# B&R Automation Studio project TD52 (part 67)

```c
  /* InitializeConditions for Delay: '<S15>/Resettable Delay' */
  Gen2_ref_DWork->icLoad_nl = true;

  /* InitializeConditions for Delay: '<Root>/Delay2' */
  Gen2_ref_DWork->icLoad_e = true;

  /* InitializeConditions for DiscreteIntegrator: '<S760>/Discrete-Time Integrator' */
  Gen2_ref_DWork->DiscreteTimeIntegrator_DSTATE_h = 1.0;

  /* InitializeConditions for Delay: '<S795>/Delay' */
  Gen2_ref_DWork->icLoad_h = true;

  /* InitializeConditions for DiscreteIntegrator: '<S579>/Discrete-Time Integrator' */
  Gen2_ref_DWork->DiscreteTimeIntegrator_DSTATE_m = 1.7;

  /* InitializeConditions for UnitDelay: '<S14>/Unit Delay4' */
  Gen2_ref_DWork->UnitDelay4_DSTATE_d = true;

  /* InitializeConditions for Delay: '<S14>/Resettable Delay2' */
  Gen2_ref_DWork->icLoad_l = true;

  /* InitializeConditions for Delay: '<S14>/Resettable Delay' */
  Gen2_ref_DWork->icLoad_i = true;

  /* InitializeConditions for UnitDelay: '<S14>/Unit Delay' */
  Gen2_ref_DWork->UnitDelay_DSTATE = 1.7;

  /* InitializeConditions for Delay: '<S14>/Resettable Delay3' */
  Gen2_ref_DWork->icLoad_f = true;

  /* InitializeConditions for DiscreteIntegrator: '<S748>/Discrete-Time Integrator' */
  Gen2_ref_DWork->DiscreteTimeIntegrator_IC_LOADI = 1U;

  /* InitializeConditions for DiscreteIntegrator: '<S748>/Discrete-Time Integrator4' */
  Gen2_ref_DWork->DiscreteTimeIntegrator4_DSTATE = 0.0;
  if (Gen2_ref_DWork->DiscreteTimeIntegrator4_DSTATE >= 0.0) {
    Gen2_ref_DWork->DiscreteTimeIntegrator4_DSTATE = 0.0;
  } else if (Gen2_ref_DWork->DiscreteTimeIntegrator4_DSTATE <= -0.3) {
    Gen2_ref_DWork->DiscreteTimeIntegrator4_DSTATE = -0.3;
  }

  /* End of InitializeConditions for DiscreteIntegrator: '<S748>/Discrete-Time Integrator4' */

  /* InitializeConditions for Delay: '<S637>/Resettable Delay' */
  Gen2_ref_DWork->icLoad_ef = true;

  /* InitializeConditions for Delay: '<S637>/Variable Integer Delay' */
  Gen2_ref_DWork->icLoad_b = true;

  /* InitializeConditions for UnitDelay: '<S628>/Unit Delay1' */
  Gen2_ref_DWork->UnitDelay1_DSTATE_a = 1.0;

  /* InitializeConditions for Delay: '<S625>/Delay' */
  Gen2_ref_DWork->Delay_DSTATE_k = 287.0;

  /* InitializeConditions for Delay: '<S666>/Resettable Delay' */
  Gen2_ref_DWork->icLoad_i0 = true;

  /* InitializeConditions for Delay: '<S714>/Resettable Delay1' */
  Gen2_ref_DWork->icLoad_np = true;

  /* InitializeConditions for Delay: '<S714>/Resettable Delay' */
  Gen2_ref_DWork->icLoad_j = true;

  /* InitializeConditions for Delay: '<S715>/Resettable Delay1' */
  Gen2_ref_DWork->icLoad_a = true;

  /* InitializeConditions for Delay: '<S715>/Resettable Delay' */
  Gen2_ref_DWork->icLoad_m3 = true;

  /* InitializeConditions for Delay: '<S431>/Delay' */
  Gen2_ref_DWork->icLoad_b3 = true;

  /* InitializeConditions for Delay: '<S78>/Variable Integer Delay' */
  Gen2_ref_DWork->icLoad_ev = true;

  /* InitializeConditions for Delay: '<S88>/Delay' */
  Gen2_ref_DWork->icLoad_d = true;

  /* InitializeConditions for Delay: '<S90>/Delay' */
  Gen2_ref_DWork->icLoad_es = true;

  /* InitializeConditions for Delay: '<S87>/Delay' */
  Gen2_ref_DWork->icLoad_evr = true;

  /* InitializeConditions for Delay: '<S89>/Delay' */
  Gen2_ref_DWork->icLoad_fg = true;

  /* InitializeConditions for Delay: '<S77>/Variable Integer Delay' */
  Gen2_ref_DWork->icLoad_c = true;

  /* InitializeConditions for Delay: '<S80>/Delay' */
  Gen2_ref_DWork->icLoad_eu = true;

  /* InitializeConditions for Delay: '<S82>/Delay' */
  Gen2_ref_DWork->icLoad_ee = true;

  /* InitializeConditions for Delay: '<S79>/Delay' */
  Gen2_ref_DWork->icLoad_ki = true;

  /* InitializeConditions for Delay: '<S81>/Delay' */
  Gen2_ref_DWork->icLoad_h3 = true;

  /* InitializeConditions for UnitDelay: '<S53>/Unit Delay4' */
  Gen2_ref_DWork->UnitDelay4_DSTATE_o = true;

  /* InitializeConditions for Delay: '<S63>/Delay' */
  Gen2_ref_DWork->icLoad_g = true;

  /* InitializeConditions for Delay: '<S64>/Delay' */
  Gen2_ref_DWork->icLoad_c1 = true;

  /* InitializeConditions for UnitDelay: '<S23>/Unit Delay3' */
  Gen2_ref_DWork->UnitDelay3_DSTATE_gf = true;

  /* InitializeConditions for DiscreteIntegrator: '<S132>/Discrete-Time Integrator' */
  Gen2_ref_DWork->DiscreteTimeIntegrator_DSTATE_g = 100000.0;

  /* InitializeConditions for Delay: '<S45>/Delay' */
  Gen2_ref_DWork->icLoad_eh = true;

  /* InitializeConditions for Delay: '<S161>/Delay2' */
  Gen2_ref_DWork->Delay2_DSTATE_f = true;

  /* InitializeConditions for DiscreteIntegrator: '<S45>/Discrete-Time Integrator1' */
  Gen2_ref_DWork->DiscreteTimeIntegrator1_IC_LOAD = 1U;

  /* InitializeConditions for Delay: '<S26>/Delay' */
  Gen2_ref_DWork->icLoad_kq = true;

  /* InitializeConditions for Delay: '<S111>/Delay2' */
  Gen2_ref_DWork->Delay2_DSTATE_k = true;

  /* InitializeConditions for DiscreteIntegrator: '<S26>/Discrete-Time Integrator' */
  Gen2_ref_DWork->DiscreteTimeIntegrator_IC_LOA_l = 1U;

  /* InitializeConditions for Delay: '<S494>/Delay' */
  Gen2_ref_DWork->icLoad_ir = true;

  /* InitializeConditions for Delay: '<S708>/Delay' */
  Gen2_ref_DWork->icLoad_nv = true;

  /* InitializeConditions for Delay: '<S524>/Delay' */
  Gen2_ref_DWork->icLoad_dk = true;

  /* InitializeConditions for Delay: '<S811>/Delay' */
  Gen2_ref_DWork->icLoad_iv = true;

  /* InitializeConditions for Delay: '<S830>/Resettable Delay' */
  Gen2_ref_DWork->icLoad_ix = true;

  /* InitializeConditions for Delay: '<S830>/Delay' */
  Gen2_ref_DWork->Delay_DSTATE_n2 = true;

  /* InitializeConditions for Delay: '<S666>/Delay' */
  Gen2_ref_DWork->Delay_DSTATE_cnq = true;

  /* InitializeConditions for Delay: '<S714>/Delay' */
  Gen2_ref_DWork->Delay_DSTATE_a = true;

  /* InitializeConditions for Delay: '<S715>/Delay' */
  Gen2_ref_DWork->Delay_DSTATE_ng = true;

  /* SystemInitialize for Atomic SubSystem: '<S418>/2nd Order Filter' */
  Gen2_ref_undOrderFilter3_Init(&Gen2_ref_DWork->undOrderFilter_j, inst);

  /* End of SystemInitialize for SubSystem: '<S418>/2nd Order Filter' */

  /* SystemInitialize for Atomic SubSystem: '<S418>/Filter' */
  /* InitializeConditions for DiscreteIntegrator: '<S439>/Discrete-Time Integrator' */
  Gen2_ref_DWork->DiscreteTimeIntegrator_IC_LOA_f = 1U;

  /* End of SystemInitialize for SubSystem: '<S418>/Filter' */

  /* SystemInitialize for Atomic SubSystem: '<S201>/Volt_filt' */
  Gen2_ref_N_TC_HP_filt_Init(&Gen2_ref_DWork->Volt_filt, inst);

  /* End of SystemInitialize for SubSystem: '<S201>/Volt_filt' */

  /* SystemInitialize for Atomic SubSystem: '<S205>/p2s_filt' */
  Gen2_ref_N_TC_HP_filt_Init(&Gen2_ref_DWork->p2s_filt, inst);

  /* End of SystemInitialize for SubSystem: '<S205>/p2s_filt' */

  /* SystemInitialize for Atomic SubSystem: '<S425>/TOF' */
  Gen2_ref_TOF_Init(&Gen2_ref_DWork->TOF_h, inst);

  /* End of SystemInitialize for SubSystem: '<S425>/TOF' */

  /* SystemInitialize for Atomic SubSystem: '<S425>/Filter' */
  /* InitializeConditions for DiscreteIntegrator: '<S485>/Discrete-Time Integrator' */
  Gen2_ref_DWork->DiscreteTimeIntegrator_IC_LOA_p = 1U;

  /* End of SystemInitialize for SubSystem: '<S425>/Filter' */

  /* SystemInitialize for Atomic SubSystem: '<S427>/TOF1' */
  Gen2_ref_TOF_Init(&Gen2_ref_DWork->TOF1_o, inst);

  /* End of SystemInitialize for SubSystem: '<S427>/TOF1' */

  /* SystemInitialize for Atomic SubSystem: '<S427>/TP' */
  Gen2_ref_TP_Init(&Gen2_ref_DWork->TP_p, inst);

  /* End of SystemInitialize for SubSystem: '<S427>/TP' */

  /* SystemInitialize for Atomic SubSystem: '<S345>/p2sfilt' */
  Gen2_ref_N_TC_HP_filt_Init(&Gen2_ref_DWork->p2sfilt, inst);

  /* End of SystemInitialize for SubSystem: '<S345>/p2sfilt' */

  /* SystemInitialize for Atomic SubSystem: '<S194>/Pel_filt' */
  Gen2_ref_N_TC_HP_filt_Init(&Gen2_ref_DWork->Pel_filt, inst);

  /* End of SystemInitialize for SubSystem: '<S194>/Pel_filt' */

  /* SystemInitialize for Atomic SubSystem: '<S875>/Pd_filt' */
  Gen2_ref_Pd_filt_Init(&Gen2_ref_DWork->Pd_filt_p, inst);

  /* End of SystemInitialize for SubSystem: '<S875>/Pd_filt' */

  /* SystemInitialize for Atomic SubSystem: '<S344>/Pd_filt' */
  Gen2_ref_Pd_filt_Init(&Gen2_ref_DWork->Pd_filt, inst);

  /* End of SystemInitialize for SubSystem: '<S344>/Pd_filt' */

  /* SystemInitialize for Atomic SubSystem: '<S344>/WO1' */
  Gen2_ref_Filter1_Init(&Gen2_ref_DWork->WO1, inst);

  /* End of SystemInitialize for SubSystem: '<S344>/WO1' */

  /* SystemInitialize for Atomic SubSystem: '<S344>/WO2' */
  Gen2_ref_Filter3_Init(Gen2_ref_ConstB.tde1, &Gen2_ref_DWork->WO2, inst);

  /* End of SystemInitialize for SubSystem: '<S344>/WO2' */

  /* SystemInitialize for Atomic SubSystem: '<S190>/N_TC_HP_filt' */
  Gen2_ref_N_TC_HP_filt_Init(&Gen2_ref_DWork->N_TC_HP_filt, inst);

  /* End of SystemInitialize for SubSystem: '<S190>/N_TC_HP_filt' */

  /* SystemInitialize for Atomic SubSystem: '<S197>/T2s_filt' */
  Gen2_ref_N_TC_HP_filt_Init(&Gen2_ref_DWork->T2s_filt, inst);

  /* End of SystemInitialize for SubSystem: '<S197>/T2s_filt' */

  /* SystemInitialize for Atomic SubSystem: '<S193>/N_TC_LP_filt' */
  Gen2_ref_N_TC_HP_filt_Init(&Gen2_ref_DWork->N_TC_LP_filt_f, inst);

  /* End of SystemInitialize for SubSystem: '<S193>/N_TC_LP_filt' */

  /* SystemInitialize for Atomic SubSystem: '<S19>/Filter1' */
  Gen2_ref_Filter3_Init(1.0, &Gen2_ref_DWork->Filter1_l, inst);

  /* End of SystemInitialize for SubSystem: '<S19>/Filter1' */

  /* SystemInitialize for Atomic SubSystem: '<S6>/TOF' */
  Gen2_ref_TOF_Init(&Gen2_ref_DWork->TOF, inst);

  /* End of SystemInitialize for SubSystem: '<S6>/TOF' */

  /* SystemInitialize for Atomic SubSystem: '<S6>/TOF1' */
  Gen2_ref_TOF_Init(&Gen2_ref_DWork->TOF1, inst);

  /* End of SystemInitialize for SubSystem: '<S6>/TOF1' */

  /* SystemInitialize for Atomic SubSystem: '<S6>/TOF2' */
  Gen2_ref_TOF_Init(&Gen2_ref_DWork->TOF2, inst);

  /* End of SystemInitialize for SubSystem: '<S6>/TOF2' */

  /* SystemInitialize for Atomic SubSystem: '<S343>/PID_Power' */
  /* InitializeConditions for DiscreteIntegrator: '<S389>/Discrete-Time Integrator' */
  Gen2_ref_DWork->DiscreteTimeIntegrator_IC_LOA_c = 1U;

  /* InitializeConditions for Delay: '<S394>/Delay' */
  Gen2_ref_DWork->icLoad_ht = true;

  /* End of SystemInitialize for SubSystem: '<S343>/PID_Power' */

  /* SystemInitialize for Atomic SubSystem: '<S760>/p2sfilt' */
  Gen2_ref_N_TC_HP_filt_Init(&Gen2_ref_DWork->p2sfilt_l, inst);

  /* End of SystemInitialize for SubSystem: '<S760>/p2sfilt' */

  /* SystemInitialize for Atomic SubSystem: '<S424>/speed Filter' */
  Gen2_ref_N_TC_HP_filt_Init(&Gen2_ref_DWork->speedFilter, inst);

  /* End of SystemInitialize for SubSystem: '<S424>/speed Filter' */

  /* SystemInitialize for Atomic SubSystem: '<S424>/Filter1' */
  Gen2_ref_Filter1_Init(&Gen2_ref_DWork->Filter1_f, inst);

  /* End of SystemInitialize for SubSystem: '<S424>/Filter1' */

  /* SystemInitialize for Atomic SubSystem: '<S761>/Filter1' */
  Gen2_ref_Filter3_Init(Gen2_ref_ConstB.Constant1_g, &Gen2_ref_DWork->Filter1_p, inst);

  /* End of SystemInitialize for SubSystem: '<S761>/Filter1' */

  /* SystemInitialize for Atomic SubSystem: '<S761>/Filter' */
  Gen2_ref_Pd_filt_Init(&Gen2_ref_DWork->Filter_kj, inst);

  /* End of SystemInitialize for SubSystem: '<S761>/Filter' */

  /* SystemInitialize for Atomic SubSystem: '<S585>/Filter1' */
  Gen2_ref_N_TC_HP_filt_Init(&Gen2_ref_DWork->Filter1_fg, inst);

  /* End of SystemInitialize for SubSystem: '<S585>/Filter1' */

  /* SystemInitialize for Atomic SubSystem: '<S585>/Filter' */
  Gen2_ref_Filter3_Init(1.0, &Gen2_ref_DWork->Filter_n, inst);

  /* End of SystemInitialize for SubSystem: '<S585>/Filter' */

  /* SystemInitialize for Atomic SubSystem: '<S306>/2nd Order Filter' */
  Gen2_ref_undOrderFilter_Init(&Gen2_ref_DWork->undOrderFilter, inst);

  /* End of SystemInitialize for SubSystem: '<S306>/2nd Order Filter' */

  /* SystemInitialize for Atomic SubSystem: '<S306>/2nd Order Filter1' */
  Gen2_ref_undOrderFilter_Init(&Gen2_ref_DWork->undOrderFilter1, inst);

  /* End of SystemInitialize for SubSystem: '<S306>/2nd Order Filter1' */

  /* SystemInitialize for Atomic SubSystem: '<S306>/2nd Order Filter2' */
  Gen2_ref_undOrderFilter_Init(&Gen2_ref_DWork->undOrderFilter2, inst);

  /* End of SystemInitialize for SubSystem: '<S306>/2nd Order Filter2' */

  /* SystemInitialize for Atomic SubSystem: '<S306>/2nd Order Filter3' */
  Gen2_ref_undOrderFilter3_Init(&Gen2_ref_DWork->undOrderFilter3, inst);

  /* End of SystemInitialize for SubSystem: '<S306>/2nd Order Filter3' */

  /* SystemInitialize for Atomic SubSystem: '<S196>/T1LP_filt' */
  Gen2_ref_N_TC_HP_filt_Init(&Gen2_ref_DWork->T1LP_filt, inst);

  /* End of SystemInitialize for SubSystem: '<S196>/T1LP_filt' */

  /* SystemInitialize for Atomic SubSystem: '<S195>/T1HP_filt' */
  Gen2_ref_N_TC_HP_filt_Init(&Gen2_ref_DWork->T1HP_filt, inst);

  /* End of SystemInitialize for SubSystem: '<S195>/T1HP_filt' */

  /* SystemInitialize for Atomic SubSystem: '<S20>/Filter1' */
  Gen2_ref_Filter3_Init(Gen2_ref_ConstB.T_filt1, &Gen2_ref_DWork->Filter1_ny, inst);

  /* End of SystemInitialize for SubSystem: '<S20>/Filter1' */

  /* SystemInitialize for Atomic SubSystem: '<S20>/Filter3' */
  Gen2_ref_Filter3_Init(Gen2_ref_ConstB.T_filt1, &Gen2_ref_DWork->Filter3_f, inst);

  /* End of SystemInitialize for SubSystem: '<S20>/Filter3' */

  /* SystemInitialize for Atomic SubSystem: '<S20>/Filter' */
  Gen2_ref_Filter3_Init(Gen2_ref_ConstB.T_filt1, &Gen2_ref_DWork->Filter_f, inst);

  /* End of SystemInitialize for SubSystem: '<S20>/Filter' */

  /* SystemInitialize for Atomic SubSystem: '<S20>/Filter2' */
  Gen2_ref_Filter3_Init(Gen2_ref_ConstB.T_filt1, &Gen2_ref_DWork->Filter2_o, inst);

  /* End of SystemInitialize for SubSystem: '<S20>/Filter2' */

  /* SystemInitialize for Atomic SubSystem: '<S14>/Filter' */
  Gen2_ref_Pd_filt_Init(&Gen2_ref_DWork->Filter_l, inst);

  /* End of SystemInitialize for SubSystem: '<S14>/Filter' */

  /* SystemInitialize for Atomic SubSystem: '<S342>/PID_Power' */
  /* InitializeConditions for DiscreteIntegrator: '<S379>/Discrete-Time Integrator' */
  Gen2_ref_DWork->DiscreteTimeIntegrator_IC_LOA_g = 1U;

  /* InitializeConditions for Delay: '<S385>/Delay' */
  Gen2_ref_DWork->icLoad_nq = true;

  /* End of SystemInitialize for SubSystem: '<S342>/PID_Power' */

  /* SystemInitialize for Atomic SubSystem: '<S737>/Filter' */
  /* InitializeConditions for DiscreteIntegrator: '<S743>/Discrete-Time Integrator' */
  Gen2_ref_DWork->DiscreteTimeIntegrator_IC_LOA_m = 1U;

  /* End of SystemInitialize for SubSystem: '<S737>/Filter' */

  /* SystemInitialize for Atomic SubSystem: '<S637>/Filter' */
  Gen2_ref_Pd_filt_Init(&Gen2_ref_DWork->Filter_bd, inst);

  /* End of SystemInitialize for SubSystem: '<S637>/Filter' */

  /* SystemInitialize for Atomic SubSystem: '<S626>/Filter1' */
  Gen2_ref_N_TC_HP_filt_Init(&Gen2_ref_DWork->Filter1_o, inst);

  /* End of SystemInitialize for SubSystem: '<S626>/Filter1' */

  /* SystemInitialize for Atomic SubSystem: '<S667>/TP' */
  Gen2_ref_TP_Init(&Gen2_ref_DWork->TP_p2, inst);

  /* End of SystemInitialize for SubSystem: '<S667>/TP' */

  /* SystemInitialize for Atomic SubSystem: '<S667>/TP1' */
  Gen2_ref_TP_Init(&Gen2_ref_DWork->TP1_c, inst);

  /* End of SystemInitialize for SubSystem: '<S667>/TP1' */

  /* SystemInitialize for Atomic SubSystem: '<S667>/TOF' */
  Gen2_ref_TOF_Init(&Gen2_ref_DWork->TOF_g, inst);

  /* End of SystemInitialize for SubSystem: '<S667>/TOF' */

  /* SystemInitialize for Atomic SubSystem: '<S630>/Filter' */
  Gen2_ref_Filter_Init(&Gen2_ref_DWork->Filter_nk, inst);

  /* End of SystemInitialize for SubSystem: '<S630>/Filter' */

  /* SystemInitialize for Atomic SubSystem: '<S636>/Filter' */
  Gen2_ref_Filter_Init(&Gen2_ref_DWork->Filter_m, inst);

  /* End of SystemInitialize for SubSystem: '<S636>/Filter' */

  /* SystemInitialize for Atomic SubSystem: '<S608>/SkipPulseWaitTP' */
  Gen2_ref_TP_Init(&Gen2_ref_DWork->SkipPulseWaitTP, inst);

  /* End of SystemInitialize for SubSystem: '<S608>/SkipPulseWaitTP' */

  /* SystemInitialize for MATLAB Function: '<S749>/MATLAB Function' */
  Gen2_ref_DWork->SR_LoadStep = true;

  /* SystemInitialize for Atomic SubSystem: '<S628>/Filter' */
  Gen2_ref_Filter3_Init(Gen2_ref_ConstB.Constant2, &Gen2_ref_DWork->Filter_b, inst);

  /* End of SystemInitialize for SubSystem: '<S628>/Filter' */

  /* SystemInitialize for Atomic SubSystem: '<S306>/2nd Order Filter4' */
  /* InitializeConditions for DiscreteIntegrator: '<S318>/Discrete-Time Integrator1' */
  Gen2_ref_DWork->DiscreteTimeIntegrator1_IC_LO_n = 1U;

  /* End of SystemInitialize for SubSystem: '<S306>/2nd Order Filter4' */

  /* SystemInitialize for Atomic SubSystem: '<S204>/p2HP_filt' */
  Gen2_ref_N_TC_HP_filt_Init(&Gen2_ref_DWork->p2HP_filt, inst);

  /* End of SystemInitialize for SubSystem: '<S204>/p2HP_filt' */

  /* SystemInitialize for Atomic SubSystem: '<S202>/p1HP_filt' */
  Gen2_ref_N_TC_HP_filt_Init(&Gen2_ref_DWork->p1HP_filt, inst);

  /* End of SystemInitialize for SubSystem: '<S202>/p1HP_filt' */

  /* SystemInitialize for MATLAB Function: '<S24>/MATLAB Function' */
  Gen2_ref_MATLABFunction_Init(&Gen2_ref_DWork->sf_MATLABFunction_f, inst);

  /* SystemInitialize for Atomic SubSystem: '<S134>/Filter' */
  Gen2_ref_Filter3_Init(Gen2_ref_ConstB.u, &Gen2_ref_DWork->Filter, inst);

  /* End of SystemInitialize for SubSystem: '<S134>/Filter' */

  /* SystemInitialize for Atomic SubSystem: '<S23>/Filter2' */
  Gen2_ref_Filter1_Init(&Gen2_ref_DWork->Filter2, inst);

  /* End of SystemInitialize for SubSystem: '<S23>/Filter2' */

  /* SystemInitialize for Atomic SubSystem: '<S23>/Filter1' */
  Gen2_ref_Filter1_Init(&Gen2_ref_DWork->Filter1, inst);

  /* End of SystemInitialize for SubSystem: '<S23>/Filter1' */

  /* SystemInitialize for Atomic SubSystem: '<S23>/Filter4' */
  Gen2_ref_Filter1_Init(&Gen2_ref_DWork->Filter4, inst);

  /* End of SystemInitialize for SubSystem: '<S23>/Filter4' */

  /* SystemInitialize for Atomic SubSystem: '<S427>/TOF3' */
  Gen2_ref_TOF_Init(&Gen2_ref_DWork->TOF3, inst);

  /* End of SystemInitialize for SubSystem: '<S427>/TOF3' */

  /* SystemInitialize for Atomic SubSystem: '<S427>/TP_ActSat_TV' */
  Gen2_ref_TP_ActSat_CBV_Init(&Gen2_ref_DWork->TP_ActSat_TV, inst);

  /* End of SystemInitialize for SubSystem: '<S427>/TP_ActSat_TV' */

  /* SystemInitialize for MATLAB Function: '<S25>/MATLAB Function' */
  Gen2_ref_MATLABFunction_Init(&Gen2_ref_DWork->sf_MATLABFunction_e, inst);

  /* SystemInitialize for Atomic SubSystem: '<S427>/TP_ActSat_CBV' */
  Gen2_ref_TP_ActSat_CBV_Init(&Gen2_ref_DWork->TP_ActSat_CBV, inst);

  /* End of SystemInitialize for SubSystem: '<S427>/TP_ActSat_CBV' */

  /* SystemInitialize for Atomic SubSystem: '<S62>/Filter3' */
  Gen2_ref_Filter3_Init(Gen2_ref_ConstB.Constant11, &Gen2_ref_DWork->Filter3, inst);

  /* End of SystemInitialize for SubSystem: '<S62>/Filter3' */

  /* SystemInitialize for Atomic SubSystem: '<S46>/cbv tracking1' */
  /* SystemInitialize for Atomic SubSystem: '<S174>/TP' */
  /* InitializeConditions for UnitDelay: '<S181>/Unit Delay2' */
  Gen2_ref_DWork->UnitDelay2_DSTATE_b = true;

  /* End of SystemInitialize for SubSystem: '<S174>/TP' */
  /* End of SystemInitialize for SubSystem: '<S46>/cbv tracking1' */

  /* SystemInitialize for Atomic SubSystem: '<S207>/p3LP_filt' */
  Gen2_ref_N_TC_HP_filt_Init(&Gen2_ref_DWork->p3LP_filt_e, inst);

  /* End of SystemInitialize for SubSystem: '<S207>/p3LP_filt' */

  /* SystemInitialize for Atomic SubSystem: '<S208>/p4LP_filt' */
  Gen2_ref_N_TC_HP_filt_Init(&Gen2_ref_DWork->p4LP_filt, inst);

  /* End of SystemInitialize for SubSystem: '<S208>/p4LP_filt' */

  /* SystemInitialize for Atomic SubSystem: '<S426>/TP' */
  Gen2_ref_TP_Init(&Gen2_ref_DWork->TP, inst);

  /* End of SystemInitialize for SubSystem: '<S426>/TP' */

  /* SystemInitialize for Atomic SubSystem: '<S426>/TP1' */
  Gen2_ref_TP_Init(&Gen2_ref_DWork->TP1, inst);

  /* End of SystemInitialize for SubSystem: '<S426>/TP1' */

  /* SystemInitialize for Atomic SubSystem: '<S192>/N_TC_LP_filt' */
  Gen2_ref_N_TC_HP_filt_Init(&Gen2_ref_DWork->N_TC_LP_filt, inst);

  /* End of SystemInitialize for SubSystem: '<S192>/N_TC_LP_filt' */

  /* SystemInitialize for Atomic SubSystem: '<S8>/Filter' */
  Gen2_ref_Pd_filt_Init(&Gen2_ref_DWork->Filter_k, inst);

  /* End of SystemInitialize for SubSystem: '<S8>/Filter' */

  /* SystemInitialize for Atomic SubSystem: '<S427>/TP_Misfire_ON' */
  Gen2_ref_TP_ActSat_CBV_Init(&Gen2_ref_DWork->TP_Misfire_ON, inst);

  /* End of SystemInitialize for SubSystem: '<S427>/TP_Misfire_ON' */

  /* SystemInitialize for Atomic SubSystem: '<S427>/TP_Misfire_OFF' */
  Gen2_ref_TP_ActSat_CBV_Init(&Gen2_ref_DWork->TP_Misfire_OFF, inst);

  /* End of SystemInitialize for SubSystem: '<S427>/TP_Misfire_OFF' */

  /* SystemInitialize for Atomic SubSystem: '<S427>/TP_Misfire_OFF1' */
  Gen2_ref_TP_ActSat_CBV_Init(&Gen2_ref_DWork->TP_Misfire_OFF1, inst);

  /* End of SystemInitialize for SubSystem: '<S427>/TP_Misfire_OFF1' */

  /* SystemInitialize for Atomic SubSystem: '<S427>/TP_Misfire_ON_2nd time' */
  Gen2_ref_TP_ActSat_CBV_Init(&Gen2_ref_DWork->TP_Misfire_ON_2ndtime, inst);

  /* End of SystemInitialize for SubSystem: '<S427>/TP_Misfire_ON_2nd time' */

  /* SystemInitialize for Atomic SubSystem: '<S427>/TP_Misfire_OFF2' */
  Gen2_ref_TP_ActSat_CBV_Init(&Gen2_ref_DWork->TP_Misfire_OFF2, inst);

  /* End of SystemInitialize for SubSystem: '<S427>/TP_Misfire_OFF2' */

  /* SystemInitialize for Atomic SubSystem: '<S19>/Filter' */
  Gen2_ref_Filter3_Init(Gen2_ref_ConstB.x0_f, &Gen2_ref_DWork->Filter_mn, inst);

  /* End of SystemInitialize for SubSystem: '<S19>/Filter' */

  /* SystemInitialize for Atomic SubSystem: '<S427>/TP_Ign retard' */
  Gen2_ref_TP_ActSat_CBV_Init(&Gen2_ref_DWork->TP_Ignretard, inst);

  /* End of SystemInitialize for SubSystem: '<S427>/TP_Ign retard' */

  /* SystemInitialize for Atomic SubSystem: '<S814>/Filter1' */
  Gen2_ref_N_TC_HP_filt_Init(&Gen2_ref_DWork->Filter1_n, inst);

  /* End of SystemInitialize for SubSystem: '<S814>/Filter1' */

  /* SystemInitialize for Atomic SubSystem: '<S831>/TP' */
  Gen2_ref_TP_Init(&Gen2_ref_DWork->TP_g, inst);

  /* End of SystemInitialize for SubSystem: '<S831>/TP' */

  /* SystemInitialize for Atomic SubSystem: '<S831>/TP1' */
  Gen2_ref_TP_Init(&Gen2_ref_DWork->TP1_l, inst);

  /* End of SystemInitialize for SubSystem: '<S831>/TP1' */

  /* SystemInitialize for Atomic SubSystem: '<S831>/TOF' */
  Gen2_ref_TOF_Init(&Gen2_ref_DWork->TOF_n, inst);

  /* End of SystemInitialize for SubSystem: '<S831>/TOF' */

  /* SystemInitialize for Atomic SubSystem: '<S8>/BDC_Trajectory' */
  /* InitializeConditions for DiscreteIntegrator: '<S417>/Discrete-Time Integrator' */
  Gen2_ref_DWork->DiscreteTimeIntegrator_DSTATE_b = 1.0;

  /* InitializeConditions for Delay: '<S434>/Delay' */
  Gen2_ref_DWork->icLoad_mu = true;

  /* SystemInitialize for Atomic SubSystem: '<S417>/p2sfilt' */
  Gen2_ref_N_TC_HP_filt_Init(&Gen2_ref_DWork->p2sfilt_b, inst);

  /* End of SystemInitialize for SubSystem: '<S417>/p2sfilt' */
  /* End of SystemInitialize for SubSystem: '<S8>/BDC_Trajectory' */

  /* SystemInitialize for Atomic SubSystem: '<S427>/TOF' */
  Gen2_ref_TOF_p_Init(&Gen2_ref_DWork->TOF_c, inst);

  /* End of SystemInitialize for SubSystem: '<S427>/TOF' */

  /* SystemInitialize for Atomic SubSystem: '<S427>/TOF2' */
  Gen2_ref_TOF_p_Init(&Gen2_ref_DWork->TOF2_d, inst);

  /* End of SystemInitialize for SubSystem: '<S427>/TOF2' */

  /* SystemInitialize for Atomic SubSystem: '<S633>/Filter' */
  Gen2_ref_Filter3_Init(Gen2_ref_ConstB.Constant3, &Gen2_ref_DWork->Filter_pj, inst);

  /* End of SystemInitialize for SubSystem: '<S633>/Filter' */

  /* SystemInitialize for Atomic SubSystem: '<S15>/Filter1' */
  Gen2_ref_N_TC_HP_filt_Init(&Gen2_ref_DWork->Filter1_fj, inst);

  /* End of SystemInitialize for SubSystem: '<S15>/Filter1' */
}

/* Model terminate function */
void Gen2_ref_terminate(RT_MODEL_Gen2_ref *const Gen2_ref_M, struct Gen2* inst)
{
  /* (no terminate code required) */
  UNUSED_PARAMETER(Gen2_ref_M);
}

/*======================== TOOL VERSION INFORMATION ==========================*
 * MATLAB 9.11 (R2021b)14-May-2021                                            *
 * Simulink 10.4 (R2021b)14-May-2021                                          *
 * Simulink Coder 9.6 (R2021b)14-May-2021                                     *
 * Embedded Coder 7.7 (R2021b)14-May-2021                                     *
 * Stateflow 10.5 (R2021b)14-May-2021                                         *
 *============================================================================*/

/*======================= LICENSE IN USE INFORMATION =========================*
 * control_toolbox                                                            *
 * matlab                                                                     *
 * matlab_coder                                                               *
 * real-time_workshop                                                         *
 * rtw_embedded_coder                                                         *
 * simulink                                                                   *
 *============================================================================*/
```
